{attribute 'enable_dynamic_creation'}
FUNCTION_BLOCK ABSTRACT FutureProcessJob EXTENDS FB_AbstructFuture IMPLEMENTS I_Observer
VAR_INPUT
END_VAR
VAR_OUTPUT
END_VAR
VAR
	_selected_future_name 	: STRING;
	_asset					: I_Asset;
	_process_job_name		: T_MaxString;
	_start_trigger_job_id	: T_MaxString;
END_VAR

PROPERTY asset : I_Asset
GET
asset := _asset;
END_GET
SET
_asset := asset;
END_SET
END_PROPERTY

METHOD execute : BOOL // Return TRUE if finish.
IF _asset = 0 THEN
	_error_id := -1;
	RETURN;
END_IF

_asset.select_process_job(_process_job_name);
_asset.set_parameters();
_asset.process_job_start();
END_METHOD

METHOD init : BOOL // Return TRUE if finish.
IF _asset = 0 THEN
	_error_id := -1;
	RETURN;
END_IF

IF _asset.set_parameters() THEN
	init := TRUE;
END_IF
END_METHOD

METHOD notify : BOOL
VAR_INPUT
	publisher	: I_Observable;
END_VAR
VAR_INST
	fb_timezone_info : FB_GetTimeZoneInformation := (bExecute := TRUE);
	text : T_MaxString;
END_VAR
VAR
	job_info : I_JobInfo;
	container : I_Container;
END_VAR
IF NOT __QUERYINTERFACE(publisher, job_info) THEN
	RETURN;
END_IF

IF 
_asset.selected_process_job.start();
END_METHOD

PROPERTY process_job_name : T_MaxString
GET
END_GET
SET
END_SET
END_PROPERTY

END_FUNCTION_BLOCK

(* stored: Version 1.1.0.1, ProductVersion 3.1.4026.17
   POU FutureProcessJob: Id {1a36e9e9-ab13-4441-b361-f9d5d764096a}, SpecialFunc None
   Property asset: Id {51a2677a-cd3d-4525-82b9-74ac378874b2}
   Get Get: Id {1890c33c-cb72-4eb7-a37d-e58b60aa543d}
   Set Set: Id {426a80f0-87db-40fd-bdb3-e036bcf06f2a}
   Method execute: Id {417962f7-daf8-4dae-990a-9d97785b54f5}
   Method init: Id {47b55248-8f59-4a6c-a73b-ca93cfa84ad7}
   Method notify: Id {314a7d2b-c7ef-495b-ac65-c73439239b8b}
   Property process_job_name: Id {7d84888d-8d41-4115-9b95-b52a582ecdf1}
   Get Get: Id {23d97b10-3316-43fb-b197-ded4fe8442d1}
   Set Set: Id {c7b02d43-d647-4f73-9553-ebc04b51e0f7} *)
